// TIA Portal project "ConveyorSystem" (V16)

(* hardware
DEVICE "HMI_1"  KTP400 Comfort
   slot 0: "HMI_1"  KTP400 Comfort  6AV2 124-2DC01-0AX0  16.0.0.0
   slot 1: "HMI_RT_1"  KTP400 Comfort  6AV2 124-2DC01-0AX0  16.0.0.0
   slot 5: "HMI_1.IE_CP_1"  PROFINET Interface  16.0.0.0
      slot 1: "PROFINET Interface_1"  PROFINET Interface
         slot 1: "Port_1"  Port
   slot 7: "HMI_1.MPI/DP_CP_1"  MPI/DP Interface  16.0.0.0
DEVICE "S7-1200 station_1"  S7-1200 Station
   slot 0: "Rack_0"  S7-1200 Rack  Rack  V1.0
   slot 1: "PLC_1"  CPU 1217C DC/DC/DC  6ES7 217-1AG40-0XB0  V4.4
   slot 2: "DI 16x24VDC_1"  6ES7 221-1BH32-0XB0  V2.0
   slot 3: "DQ 16x24VDC_1"  SM 1222 DQ16 x 24VDC  6ES7 222-1BH32-0XB0  V2.0
*)

// ===== PLC "PLC_1"  CPU 1217C DC/DC/DC =====

VAR_GLOBAL   // PLC tag table "Default tag table"
   "System_Byte" AT %MB1 : Byte;
   "FirstScan" AT %M1.0 : Bool;
   "DiagStatusUpdate" AT %M1.1 : Bool;
   "AlwaysTRUE" AT %M1.2 : Bool;
   "AlwaysFALSE" AT %M1.3 : Bool;
   "Clock_Byte" AT %MB0 : Byte;
   "Clock_10Hz" AT %M0.0 : Bool;
   "Clock_5Hz" AT %M0.1 : Bool;
   "Clock_2.5Hz" AT %M0.2 : Bool;
   "Clock_2Hz" AT %M0.3 : Bool;
   "Clock_1.25Hz" AT %M0.4 : Bool;
   "Clock_1Hz" AT %M0.5 : Bool;
   "Clock_0.625Hz" AT %M0.6 : Bool;
   "Clock_0.5Hz" AT %M0.7 : Bool;
END_VAR

VAR_GLOBAL   // PLC tag table "Di"
   "Coveyor_Di" AT %I0.0 : "tyDi";
END_VAR

VAR_GLOBAL   // PLC tag table "Do"
   "ConveyorDo" AT %Q0.0 : "tyOutputs";
END_VAR

VAR_GLOBAL   // PLC tag table "SmemaIn"
   "SmemaIn-ReadyToSend" AT %I2.0 : Bool;
   "SmemaIn-ReadyToRecive" AT %Q2.0 : Bool;
END_VAR

VAR_GLOBAL   // PLC tag table "SmemaOut"
   "SmemaOut-ReadyToRecive" AT %I2.1 : Bool;
   "SmemaOut-ReadyToSend" AT %Q2.1 : Bool;
END_VAR

// folder: HmiExchange

TYPE "TyStopperHmiDataExchange"
   STRUCT
      FromPlcToHmi : Struct
         StopperUp : Bool;
         StopperDown : Bool;
         ProductPresent_BufferSpace : Bool;
         ProductPresent_Stopper : Bool;
      END_STRUCT;
      FromHmiToPlc : Struct
         DoStopperUp : Bool;
      END_STRUCT;
   END_STRUCT;
END_TYPE

TYPE "tyHmiMotorControl"
VERSION : 0.1
   STRUCT
      DataHmiToPlc : Struct
         doStartMotorForward : Bool;
      END_STRUCT;
      DataPlcToHmi : Struct
         MotorIsRuning : Bool;
      END_STRUCT;
   END_STRUCT;
END_TYPE

TYPE "TyModeControl"
VERSION : 0.1
   STRUCT
      StopPushButton : Bool;
      StartPusbutton : Bool;
      ManualMode : Bool;
      Reset : Bool;
   END_STRUCT;
END_TYPE

// folder: IO

TYPE "tyDi"
   STRUCT
      "IT-1-S1" : Bool;   // Input Trigger
      "B1-S1" : Bool;   // Buffer product detected
      "ST1-S1" : Bool;   // Stopper Up
      "ST1-S2" : Bool;   // Stopper Down
      "ST1-S3" : Bool;   // Stopper product detected
      "B2-S2" : Bool;   // Buffer product detected
      "ST2-S1" : Bool;   // Stopper Up
      "ST2-S2" : Bool;   // Stopper Down
      "ST2-S3" : Bool;   // Stopper product detected
      "IT2-S1" : Bool;   // Product Ready Acc
      "OT1-S1" : Bool;   // Output Trigger
      "M1-Runing" : Bool;   // Motor Forward Feedback
      MotorTemp_Ok : Bool;
      MotorProtection_Ok : Bool;
      "E-Stop_Ok" : Bool;
      AirSupply_Ok : Bool;
   END_STRUCT;
END_TYPE

TYPE "tyOutputs"
VERSION : 0.1
   STRUCT
      MotorForward : Bool;   // MotorForward
      "ST1-V1" : Bool;   // Stopper Valve
      "ST2-V1" : Bool;   // Stopper Valve
      ProductOnWorkPossition : Bool;
   END_STRUCT;
END_TYPE

// folder: (top level)

DATA_BLOCK "GVL"   // DB1
{ S7_Optimized_Access := 'TRUE' }
VERSION : 0.1
   VAR
      TestModeStruct : Struct
         TestMode : Bool;
      END_STRUCT;
      ScreenMode : Struct
         CurrentScreen : Int;
      END_STRUCT;
   END_VAR
   VAR RETAIN
      Parameters : Struct
         AccModeSellected : Bool;
         CurrentMode : Int;
      END_STRUCT;
   END_VAR
   VAR
      JobMailBox : Array[0..3] of Word;
      ScreenNumberHmiControl : Int;
      HmiCurrentScreenNumber : Array[0..4] of Word;
      CurrentScreen : Int;
   END_VAR
BEGIN
   JobMailBox[0] := 51;
   JobMailBox[2] := 0;
   JobMailBox[3] := 0;
END_DATA_BLOCK

// folder: DB

DATA_BLOCK "MainBlock_DB"   // DB2
{ S7_Optimized_Access := 'TRUE' }
VERSION : 0.1
// stored: InstanceOfName MainBlock
"MainBlock"
BEGIN
END_DATA_BLOCK

// folder: (top level)

ORGANIZATION_BLOCK "Main"   // OB1, LAD, ProgramCycle
TITLE = "Main Program Sweep (Cycle)"
{ S7_Optimized_Access := 'TRUE' }
VERSION : 0.1
   VAR_INPUT
      Initial_Call : Bool;   // Initial call of this OB
      Remanence : Bool;   // =True, if remanent data are available
   END_VAR
BEGIN

REGION Network 1
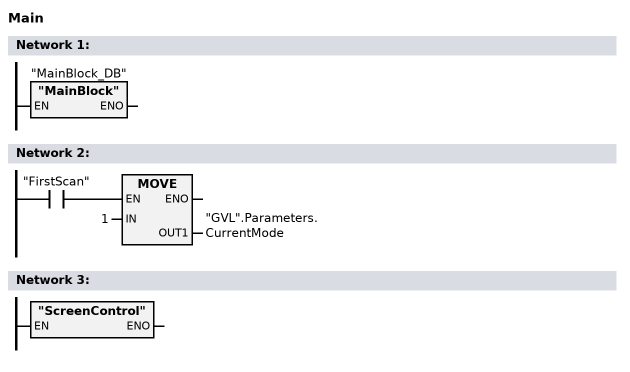
   RUNG wire#powerrail
      "MainBlock_DB"()
   END_RUNG
   // the same network as SCL:
   "MainBlock_DB"();   // "MainBlock"
END_REGION

REGION Network 2
   RUNG wire#powerrail
      Contact( "FirstScan" )
      Move(in := 1, out1 => "GVL".Parameters.CurrentMode)
   END_RUNG
   // the same network as SCL:
   IF "FirstScan" THEN "GVL".Parameters.CurrentMode := 1; END_IF;
END_REGION

REGION Network 3
   RUNG wire#powerrail
      "ScreenControl"()
   END_RUNG
   // the same network as SCL:
   "ScreenControl"();
END_REGION
END_ORGANIZATION_BLOCK

// folder: Devices

FUNCTION_BLOCK "Stopper"   // FB1, SCL
{ S7_Optimized_Access := 'TRUE' }
VERSION : 0.1
   VAR_INPUT
      TestMode : Bool;
      Di_Activate_StopperUp : Bool;
      Di_StopperSensorUp : Bool;
      Di_StopperSensorDown : Bool;
      Di_StopperSensorProductDetected : Bool;
      Di_BufferrSensorProductDetected : Bool;
      ManualMode : Bool;
   END_VAR
   VAR_OUTPUT
      Do_Fault : Bool;
      Do_OutputSolenoidValve_Up : Bool;
      Do_StopperIsUp : Bool;
      Do_StopperIsDown : Bool;
      Do_ProductDetectedStopper : Bool;
      Do_ProductDetectedBuffer : Bool;
   END_VAR
   VAR
      HmiStopperExchange : "TyStopperHmiDataExchange";
      StopperUpFault : TON_TIME;
      StopperDownFault : TON_TIME;
   END_VAR
BEGIN
   //=============================================================================
   // Dmitri Raihtsaum - Copyright 2024
   // Created By: Dmitri Raihtsaum
   //-----------------------------------------------------------------------------
   // Tested with:   6ES7 217-1AG40-0XB0
   // Engineering:   TIA Portal V16
   // Functionality:  Stopper Controll fucntion block
   // Date: 13.10.2024
   // Rev 0.1
   //=============================================================================

   //Manual Auto Control Switch
   IF #ManualMode THEN
       IF #HmiStopperExchange.FromHmiToPlc.DoStopperUp THEN
           #Do_OutputSolenoidValve_Up := TRUE;
       ELSE
           #Do_OutputSolenoidValve_Up := FALSE;
       END_IF;
   ELSE
       IF #Di_Activate_StopperUp THEN
           #Do_OutputSolenoidValve_Up := TRUE;
       ELSE
           #Do_OutputSolenoidValve_Up := FALSE;
       END_IF;
   END_IF;

   //Fault Control
   IF #TestMode THEN
       #StopperUpFault(IN := FALSE,
                       PT := t#0ms);
       #StopperDownFault(IN := FALSE,
                         PT := t#0ms);
   ELSE
       #StopperUpFault(IN := #Di_Activate_StopperUp AND NOT #Do_StopperIsUp,
                       PT := t#2s);
       #StopperDownFault(IN := NOT #Di_Activate_StopperUp AND NOT #Do_StopperIsDown,
                         PT := t#2s);
   END_IF;

   //Fault Control
   IF #StopperDownFault.Q OR #StopperUpFault.Q THEN
       #Do_Fault := TRUE;
   ELSE
       #Do_Fault := FALSE;
   END_IF;

   //Do
   IF #TestMode THEN
       #Do_StopperIsUp := #Do_OutputSolenoidValve_Up;
       #Do_StopperIsDown := NOT  #Do_OutputSolenoidValve_Up;
   ELSE
       #Do_StopperIsUp := #Di_StopperSensorUp;
       #Do_StopperIsDown := #Di_StopperSensorDown;
   END_IF;
   #Do_ProductDetectedStopper := #Di_StopperSensorProductDetected;
   #Do_ProductDetectedBuffer := #Di_BufferrSensorProductDetected;

   //Hmi
   #HmiStopperExchange.FromPlcToHmi.StopperUp := #Do_StopperIsUp;
   #HmiStopperExchange.FromPlcToHmi.StopperDown := #Do_StopperIsDown;
   #HmiStopperExchange.FromPlcToHmi.ProductPresent_BufferSpace := #Di_StopperSensorProductDetected;
   #HmiStopperExchange.FromPlcToHmi.ProductPresent_Stopper := #Di_BufferrSensorProductDetected;

   //=============================================================================
   //END
   //=============================================================================
END_FUNCTION_BLOCK

FUNCTION_BLOCK "MotorControl"   // FB2, SCL
{ S7_Optimized_Access := 'TRUE' }
VERSION : 0.1
   VAR_INPUT
      TestMode : Bool;
      ManualMode : Bool;
      Di_doStartMotorForward : Bool;
      Di_MotorForwardFeedback : Bool;
      Di_MotorTemp_Ok : Bool;
      Di_MotorProtection_Ok : Bool;
   END_VAR
   VAR_OUTPUT
      Do_Fault : Bool;
      Do_StartMotorForward : Bool;
      Do_MotorIsRuning : Bool;
   END_VAR
   VAR
      Hmi_MotorDataExchange : "tyHmiMotorControl";
      MotorRunFault : TON_TIME;
      MotorStopFault : TON_TIME;
   END_VAR
BEGIN
   //=============================================================================
   // Dmitri Raihtsaum - Copyright 2024
   // Created By: Dmitri Raihtsaum
   //-----------------------------------------------------------------------------
   // Tested with:   6ES7 217-1AG40-0XB0 
   // Engineering:   TIA Portal V16
   // Functionality:  Motor Controll fucntion block
   // Date: 13.10.2024
   // Rev 0.1
   //=============================================================================

   //Manual Auto Control Switch
   IF #ManualMode THEN
       IF #Hmi_MotorDataExchange.DataHmiToPlc.doStartMotorForward THEN
           #Do_StartMotorForward := TRUE;
       ELSE
           #Do_StartMotorForward := FALSE;
       END_IF;
   ELSE
       IF #Di_doStartMotorForward THEN
           #Do_StartMotorForward := TRUE;
       ELSE
           #Do_StartMotorForward := FALSE;
       END_IF;
   END_IF;
   //Fault Control
   IF #TestMode THEN
       #MotorRunFault(IN := FALSE,
                      PT := T#2s);
       #MotorStopFault(IN := FALSE,
                       PT := T#2s);
   ELSE
       #MotorRunFault(IN := #Di_doStartMotorForward AND NOT #Di_MotorForwardFeedback,
                      PT := T#2s);
       #MotorStopFault(IN := NOT #Di_doStartMotorForward AND #Di_MotorForwardFeedback,
                       PT := T#2s);
   END_IF;
   //Fault Control
   IF NOT #TestMode THEN
       #Do_Fault := NOT #Di_MotorTemp_Ok OR NOT #Di_MotorProtection_Ok OR #MotorRunFault.Q OR #MotorStopFault.Q;
   ELSE
       #Do_Fault := FALSE;
   END_IF;
   //Motor Feedback 
   IF NOT #TestMode THEN
       #Do_MotorIsRuning := #Di_MotorForwardFeedback;
   ELSE
       #Do_MotorIsRuning := #Do_StartMotorForward;
   END_IF;

   #Hmi_MotorDataExchange.DataPlcToHmi.MotorIsRuning := #Do_MotorIsRuning;

   //=============================================================================
   //END
   //=============================================================================
END_FUNCTION_BLOCK

// folder: Logic

FUNCTION_BLOCK "SystemControl"   // FB3, SCL
{ S7_Optimized_Access := 'TRUE' }
VERSION : 0.1
   VAR_INPUT
      Di_ReadyToStop : Bool;
      Di_ExternalFault : Bool;
   END_VAR
   VAR_OUTPUT
      SystemStateOutput : Int;
      Do_ManualMode : Bool;
      Do_Reset : Bool;
   END_VAR
   VAR
      CurrentState : Int;
      HmiSystemControl : "TyModeControl";
      StopTimer : TON_TIME;
   END_VAR
BEGIN
   //=============================================================================
   // Dmitri Raihtsaum - Copyright 2024
   // Created By: Dmitri Raihtsaum
   //-----------------------------------------------------------------------------
   // Tested with:   6ES7 215-1AG40-0XB0
   // Engineering:   TIA Portal V16
   // Functionality:  Mode Control 
   // Date: 13.10.2024
   // Rev 0.1
   //=============================================================================

   CASE #CurrentState OF
       0:  // Var Init
           IF "FirstScan" OR #HmiSystemControl.Reset THEN
               #CurrentState := 1;
           END_IF;

       1:  // Stop
           IF #HmiSystemControl.StartPusbutton THEN
               #CurrentState := 2;
           END_IF;

       2: //AutoRun
           IF (#HmiSystemControl.StopPushButton AND NOT #Di_ReadyToStop) THEN
               #CurrentState := 3;
           ELSIF (#HmiSystemControl.StopPushButton AND #Di_ReadyToStop) THEN
               #CurrentState := 1;
           END_IF;

       3: //AutoStop
           IF #Di_ReadyToStop OR #StopTimer.Q THEN
               #CurrentState := 1;
           END_IF;
   END_CASE;

   #StopTimer(IN := #HmiSystemControl.StopPushButton,
              PT := T#2s);

   IF #Di_ExternalFault THEN
       #CurrentState := 0;
   END_IF;
   #Do_ManualMode := #HmiSystemControl.ManualMode;

   #SystemStateOutput := #CurrentState;

   //=============================================================================
   //END
   //=============================================================================
END_FUNCTION_BLOCK

FUNCTION_BLOCK "MainBlock"   // FB4, SCL
{ S7_Optimized_Access := 'TRUE' }
VERSION : 0.1
   VAR
      MainLogic_Instance : "MainLogic";
   END_VAR
BEGIN
   //=============================================================================
   // Dmitri Raihtsaum - Copyright 2024
   // Created By: Dmitri Raihtsaum
   //-----------------------------------------------------------------------------
   // Tested with:   6ES7 217-1AG40-0XB0 
   // Engineering:   TIA Portal V16
   // Functionality:  Main Block Logic
   // Date: 13.10.2024
   // Rev 0.1
   //=============================================================================
   //
   CASE "GVL".Parameters.CurrentMode OF
       1:  // Mode 1
           #MainLogic_Instance(Di_Input:="Coveyor_Di",
                               "SmemaIn-ReadyToSend":="SmemaIn-ReadyToSend",
                               "SmemaOut-ReadyToRecive":="SmemaOut-ReadyToRecive",
                               TestMode:="GVL".TestModeStruct.TestMode,
                               Do_Output=>"ConveyorDo",
                               "SmemaIn-ReadyToRecive"=>"SmemaIn-ReadyToRecive",
                               "SmemaOut-ReadyToSend"=>"SmemaOut-ReadyToSend");

       2:  // Mode 2
           ;

   END_CASE;

   //=============================================================================
   //END
   //=============================================================================
END_FUNCTION_BLOCK

FUNCTION_BLOCK "MainLogic"   // FB5, SCL
{ S7_Optimized_Access := 'TRUE' }
VERSION : 0.1
   VAR_INPUT
      Di_Input : "tyDi";
      "SmemaIn-ReadyToSend" : Bool;
      "SmemaOut-ReadyToRecive" : Bool;
      TestMode : Bool;
      OperatorOrRobotAcknowledge_Setting : Bool;
   END_VAR
   VAR_OUTPUT
      Do_Output : "tyOutputs";
      "SmemaIn-ReadyToRecive" : Bool := false;
      "SmemaOut-ReadyToSend" : Bool := false;
      GlobalReset : Bool := false;
      Alarms0 : Word := 16#0;
   END_VAR
   VAR
      CurrentState : Int;
      Stopper_1 : "Stopper";
      Stopper_2 : "Stopper";
      MotorControl_1 : "MotorControl";
      SystemControl_Instance : "SystemControl";
      StepTimer1 : TON_TIME;
      StepTimer2 : TON_TIME;
      OutputTriggerDelay : TOF_TIME;
   END_VAR
BEGIN
   //=============================================================================
   // Dmitri Raihtsaum - Copyright 2024
   // Created By: Dmitri Raihtsaum
   //-----------------------------------------------------------------------------
   // Tested with:   6ES7 217-1AG40-0XB0 
   // Engineering:   TIA Portal V16
   // Functionality:  Main Logic
   // Date: 13.10.2024
   // Rev 0.1
   //=============================================================================

   CASE #CurrentState OF
       0:  // Var Init
           #StepTimer1(IN:=FALSE,
                       PT:=T#0ms);
           #StepTimer2(IN:=FALSE,
                       PT:=T#0ms);
           #"SmemaIn-ReadyToRecive" := FALSE;
           #"SmemaOut-ReadyToSend" := FALSE;
           #Do_Output.ProductOnWorkPossition := FALSE;
           #Stopper_1.Di_Activate_StopperUp := TRUE;
           #Stopper_2.Di_Activate_StopperUp := TRUE;
           #MotorControl_1.Di_doStartMotorForward := FALSE;
           #SystemControl_Instance.Di_ReadyToStop := TRUE;
           IF #SystemControl_Instance.SystemStateOutput = 2 THEN
               #CurrentState := 1;
           END_IF;

       1:  // Stopper Test 
           #Stopper_1.Di_Activate_StopperUp := FALSE;
           #Stopper_2.Di_Activate_StopperUp := FALSE;
           #StepTimer1(IN := TRUE,
                       PT := T#700ms);
           #StepTimer2(IN := FALSE,
                       PT := T#0ms);
           IF #StepTimer1.Q THEN
               #CurrentState := 2;
           END_IF;
       2: // Stopper Test 
           #StepTimer1(IN := FALSE,
                       PT := T#0ms);
           #StepTimer2(IN := TRUE,
                       PT := T#500ms);
           #Stopper_1.Di_Activate_StopperUp := TRUE;
           #Stopper_2.Di_Activate_StopperUp := TRUE;
           IF #StepTimer2.Q THEN
               #CurrentState := 3;
           END_IF;

       3:// Stopper Test 
           #StepTimer1(IN := TRUE,
                       PT := T#1s);
           #StepTimer2(IN := FALSE,
                       PT := T#0ms);
           #MotorControl_1.Di_doStartMotorForward := TRUE;
           IF #StepTimer1.Q THEN
               #CurrentState := 10;
           END_IF;

       6: //Idle 
           #StepTimer1(IN := FALSE,
                       PT := T#0ms);
           #StepTimer2(IN := FALSE,
                       PT := T#0ms);
           #"SmemaIn-ReadyToRecive" := FALSE;
           #"SmemaOut-ReadyToSend" := FALSE;
           #Do_Output.ProductOnWorkPossition := FALSE;
           #Stopper_1.Di_Activate_StopperUp := TRUE;
           #Stopper_2.Di_Activate_StopperUp := TRUE;
           #MotorControl_1.Di_doStartMotorForward := FALSE;
           #SystemControl_Instance.Di_ReadyToStop := TRUE;
           // Product move sellection 
           IF #SystemControl_Instance.SystemStateOutput = 2 THEN
               IF (#"SmemaIn-ReadyToSend" OR #Di_Input."IT-1-S1") AND NOT #Stopper_1.Do_ProductDetectedStopper THEN
                   #CurrentState := 10;
               ELSIF NOT #Stopper_2.Do_ProductDetectedStopper AND #Stopper_1.Do_ProductDetectedStopper THEN
                   #CurrentState := 30;
               ELSIF #OperatorOrRobotAcknowledge_Setting AND #Stopper_2.Do_ProductDetectedStopper AND #"SmemaOut-ReadyToRecive" AND #Di_Input."IT2-S1"
               THEN
                   #CurrentState := 40;
               ELSIF NOT #OperatorOrRobotAcknowledge_Setting AND #Stopper_2.Do_ProductDetectedStopper AND #"SmemaOut-ReadyToRecive" THEN
                   #CurrentState := 40;
               END_IF;
           END_IF;


       10: // Pass sellection - Go to buffer 1 - or move to buffer 2 
           #SystemControl_Instance.Di_ReadyToStop := FALSE;
           IF NOT #Stopper_2.Do_ProductDetectedStopper AND NOT #"SmemaOut-ReadyToRecive" AND NOT #OperatorOrRobotAcknowledge_Setting THEN
               #CurrentState := 20;
           ELSIF NOT #Stopper_2.Do_ProductDetectedStopper AND #"SmemaOut-ReadyToRecive" AND NOT #OperatorOrRobotAcknowledge_Setting THEN
               #CurrentState := 50;
           ELSE
               #CurrentState := 11;
           END_IF;

       11: // Move to stopper 1
           #SystemControl_Instance.Di_ReadyToStop := FALSE;
           #StepTimer1(IN := FALSE,
                       PT := T#0ms);
           #StepTimer2(IN := FALSE,
                       PT := T#0ms);
           #"SmemaIn-ReadyToRecive" := TRUE;
           #Stopper_1.Di_Activate_StopperUp := TRUE;
           #MotorControl_1.Di_doStartMotorForward := TRUE;
           IF #Stopper_1.Do_ProductDetectedStopper THEN
               #CurrentState := 12;
           END_IF;

       12: // Stop product to stopper 1
           #StepTimer1(IN := TRUE,
                       PT := T#1s);
           #StepTimer2(IN := FALSE,
                       PT := T#0ms);
           #"SmemaIn-ReadyToRecive" := FALSE;
           #Stopper_1.Di_Activate_StopperUp := TRUE;
           #MotorControl_1.Di_doStartMotorForward := FALSE;
           IF #StepTimer1.Q THEN
               #CurrentState := 6;
           END_IF;

       20: // Move to stopper 2
           #SystemControl_Instance.Di_ReadyToStop := FALSE;
           #StepTimer1(IN := FALSE,
                       PT := T#0ms);
           #StepTimer2(IN := FALSE,
                       PT := T#0ms);
           #"SmemaIn-ReadyToRecive" := TRUE;
           #Stopper_1.Di_Activate_StopperUp := FALSE;
           #Stopper_2.Di_Activate_StopperUp := TRUE;
           #MotorControl_1.Di_doStartMotorForward := TRUE;
           IF #Stopper_2.Do_ProductDetectedStopper THEN
               #CurrentState := 21;
           END_IF;

       21: // Stop product to stopper 2
           #StepTimer1(IN := TRUE,
                       PT := T#1s);
           #StepTimer2(IN := FALSE,
                       PT := T#0ms);
           #"SmemaIn-ReadyToRecive" := FALSE;
           #Stopper_1.Di_Activate_StopperUp := TRUE;
           #Stopper_2.Di_Activate_StopperUp := TRUE;
           #MotorControl_1.Di_doStartMotorForward := FALSE;
           IF #StepTimer1.Q THEN
               #CurrentState := 6;
           END_IF;

       30 : //  Buffer 1 to buffer 2 transit 
           #SystemControl_Instance.Di_ReadyToStop := FALSE;
           #StepTimer1(IN := FALSE,
                       PT := T#0ms);
           #StepTimer2(IN := FALSE,
                       PT := T#0ms);
           #Stopper_1.Di_Activate_StopperUp := FALSE;
           #Stopper_2.Di_Activate_StopperUp := TRUE;
           #MotorControl_1.Di_doStartMotorForward := TRUE;
           IF #Stopper_2.Do_ProductDetectedStopper THEN
               #CurrentState := 31;
           END_IF;

       31: // Buffer 1 to buffer 2 transit 
           #StepTimer1(IN := TRUE,
                       PT := T#1s);
           #StepTimer2(IN := FALSE,
                       PT := T#0ms);
           #Stopper_1.Di_Activate_StopperUp := TRUE;
           #Stopper_2.Di_Activate_StopperUp := TRUE;
           #MotorControl_1.Di_doStartMotorForward := FALSE;
           IF #StepTimer1.Q THEN
               #CurrentState := 6;
           END_IF;

       40 : // Out Transit 
           #SystemControl_Instance.Di_ReadyToStop := FALSE;
           #OutputTriggerDelay(IN:=FALSE,
                               PT:=T#0ms);
           #Stopper_2.Di_Activate_StopperUp := FALSE;
           #MotorControl_1.Di_doStartMotorForward := TRUE;
           IF #Di_Input."OT1-S1" THEN
               #CurrentState := 41;
           END_IF;

       41: //  Out Transit 
           #OutputTriggerDelay(IN := #Di_Input."OT1-S1",
                               PT := T#15s);
           IF #OutputTriggerDelay.ET > T#6s THEN
               #CurrentState := 6;
           END_IF;


       50: // Transit withour stopper 
           #SystemControl_Instance.Di_ReadyToStop := FALSE;
           #StepTimer1(IN := FALSE,
                       PT := T#0ms);
           #StepTimer2(IN := FALSE,
                       PT := T#0ms);
           #OutputTriggerDelay(IN := FALSE,
                               PT := T#0ms);
           #Stopper_1.Di_Activate_StopperUp := FALSE;
           #Stopper_2.Di_Activate_StopperUp := FALSE;
           #MotorControl_1.Di_doStartMotorForward := TRUE;
           IF #Di_Input."OT1-S1" THEN
               #CurrentState := 51;
           END_IF;

       51: // Transit withour stopper 
           #OutputTriggerDelay(IN := #Di_Input."OT1-S1",
                               PT := T#15s);
           IF #OutputTriggerDelay.ET > T#6s THEN
               #CurrentState := 6;
           END_IF;


   END_CASE;

   IF #SystemControl_Instance.CurrentState < 2 THEN
       #CurrentState := 6;
   END_IF;

   #Stopper_1(TestMode:=#TestMode,
              Di_StopperSensorUp:=#Di_Input."ST1-S1",
              Di_StopperSensorDown:=#Di_Input."ST1-S2",
              Di_StopperSensorProductDetected:=#Di_Input."ST1-S3",
              Di_BufferrSensorProductDetected:=#Di_Input."B1-S1",
              ManualMode:=#SystemControl_Instance.Do_ManualMode,
              Do_OutputSolenoidValve_Up=>#Do_Output."ST1-V1");
   #Stopper_2(TestMode:=#TestMode,
              Di_StopperSensorUp:=#Di_Input."ST2-S1",
              Di_StopperSensorDown:=#Di_Input."ST2-S2",
              Di_StopperSensorProductDetected:=#Di_Input."ST2-S3",
              Di_BufferrSensorProductDetected:=#Di_Input."B2-S2",
              ManualMode:=#SystemControl_Instance.Do_ManualMode,
              Do_OutputSolenoidValve_Up=>#Do_Output."ST2-V1");
   #MotorControl_1(TestMode:=#TestMode,
                   ManualMode:=#SystemControl_Instance.Do_ManualMode,
                   Di_MotorForwardFeedback:=#Di_Input."M1-Runing",
                   Di_MotorTemp_Ok:=#Di_Input.MotorTemp_Ok,
                   Di_MotorProtection_Ok:=#Di_Input.MotorProtection_Ok,
                   Do_StartMotorForward=>#Do_Output.MotorForward);
   #SystemControl_Instance();

   REGION Alarms
       IF #TestMode THEN
           #Alarms0.%X0 := FALSE;
           #Alarms0.%X1 := FALSE;
           #Alarms0.%X2 := FALSE;
           #Alarms0.%X3 := FALSE;
           #Alarms0.%X4 := FALSE;
           #Alarms0.%X5 := FALSE;
           #Alarms0.%X6 := FALSE;
           //  #Alarms0.%X7 :=
       ELSE

           #Alarms0.%X0 := NOT #Di_Input.MotorTemp_Ok;
           #Alarms0.%X1 := NOT #Di_Input.MotorProtection_Ok;
           #Alarms0.%X2 := NOT #Di_Input."E-Stop_Ok";
           #Alarms0.%X3 := NOT #Di_Input.AirSupply_Ok;
           #Alarms0.%X4 := #Stopper_1.Do_Fault;
           #Alarms0.%X5 := #Stopper_1.Do_Fault;
           #Alarms0.%X6 := #MotorControl_1.Do_Fault;
           //  #Alarms0.%X7 :=
       END_IF;

   END_REGION
   //=============================================================================
   //END
   //=============================================================================
END_FUNCTION_BLOCK

FUNCTION "ScreenControl" : Void   // FC1, SCL
{ S7_Optimized_Access := 'TRUE' }
VERSION : 0.1
BEGIN
   //=============================================================================
   // Dmitri Raihtsaum - Copyright 2024
   // Created By: Dmitri Raihtsaum
   //-----------------------------------------------------------------------------
   // Tested with:   6ES7 217-1AG40-0XB0 
   // Engineering:   TIA Portal V16
   // Functionality:  Screen Control
   // Date: 13.10.2024
   // Rev 0.1
   //=============================================================================

   "GVL".CurrentScreen := WORD_TO_INT("GVL".HmiCurrentScreenNumber[1]); // Recive information from current screen 
   "GVL".ScreenNumberHmiControl := "GVL".Parameters.CurrentMode * 10; // Prepare variable to activate screen

   IF "GVL".CurrentScreen / 10 <> "GVL".Parameters.CurrentMode THEN // Compare current screen and current mode
       "GVL".JobMailBox[1] := INT_TO_WORD("GVL".ScreenNumberHmiControl); // Send screen number to hmi to change screen 
       "GVL".JobMailBox[0] := 16#33; // Jobmailbox adress
       "GVL".JobMailBox[2] := 16#00; // Not used 
       "GVL".JobMailBox[3] := 16#00; // Not used 
   END_IF;

   //=============================================================================
   //END
   //=============================================================================
END_FUNCTION

(* ===== HMI "HMI_RT_1" =====
system functions are stored by id; their names below are inferred from use
connection "HMI_Connection_1": ETHERNET, S7_1200_OMS

HMI tags "Di"
   "Di" : tyDi = PLC Coveyor_Di AT %I0.0, 1 s

HMI tags "Do"
   "Do" : tyOutputs = PLC ConveyorDo AT %Q0.0, 1 s

HMI tags "SmemaIn"
   "SmemaIn-ReadyToRecive" : Bool = PLC "SmemaIn-ReadyToRecive" AT %Q2.0, 1 s
   "SmemaIn-ReadyToSend" : Bool = PLC "SmemaIn-ReadyToSend" AT %I2.0, 1 s

HMI tags "SmemaOut"
   "SmemaOut-ReadyToRecive" : Bool = PLC "SmemaOut-ReadyToRecive" AT %I2.1, 1 s
   "SmemaOut-ReadyToSend" : Bool = PLC "SmemaOut-ReadyToSend" AT %Q2.1, 1 s

HMI tags "SystemControl"
   "HmiSystemControl" : TyModeControl = PLC MainBlock_DB.MainLogic_Instance.SystemControl_Instance.HmiSystemControl, 1 s

HMI tags "Stoppers"
   "HmiStopperExchange1" : TyStopperHmiDataExchange = PLC MainBlock_DB.MainLogic_Instance.Stopper_1.HmiStopperExchange, 1 s
   "HmiStopperExchange2" : TyStopperHmiDataExchange = PLC MainBlock_DB.MainLogic_Instance.Stopper_2.HmiStopperExchange, 1 s

HMI tags "Motors"
   "Hmi_MotorDataExchange" : tyHmiMotorControl = PLC MainBlock_DB.MainLogic_Instance.MotorControl_1.Hmi_MotorDataExchange, 1 s

HMI tags "Parameters"
   "CurrentModeSellection" : Int = PLC GVL.Parameters.CurrentMode, 1 s
   "AccModeActivated" : Bool = PLC GVL.Parameters.AccModeSellected AT %DB1.DBW0, 1 s

HMI tags "SystemData"
   "SystemMode" : Int = PLC MainBlock_DB.MainLogic_Instance.SystemControl_Instance.SystemStateOutput, 1 s

HMI tags "Alarm0"
   "Alarm0" : Word = PLC MainBlock_DB.MainLogic_Instance.Alarms0 AT %DB1.DBW0, 1 s

discrete alarms
   1: 'Motor Temperature fault', class Errors, trigger "Alarm0" bit 0
   2: 'Motor Protection Triggered', class Errors, trigger "Alarm0" bit 1
   3: 'E-Stop Triggred', class Errors, trigger "Alarm0" bit 2
   4: 'Air Sypply Fault', class Errors, trigger "Alarm0" bit 3
   5: 'Stopper 1 Fault', class Errors, trigger "Alarm0" bit 4
   6: 'Stopper 2 Fault', class Errors, trigger "Alarm0" bit 5
   7: 'Motor Fault', class Errors, trigger "Alarm0" bit 6

Template "Template_1" 480x272
   Button "Template_Button_1" at 12,7 size 96x32; TextOff 'Start'
      ObjectEnable <- "ManualMode"
      on Press: function_b14e0dd5("StartPusbutton", 0); ResetBit("doStartMotorForward"); ResetBit("DoStopperUp"); ResetBit("DoStopperUp")
      Appearance <- "SystemMode"
   Button "Template_Button_2" at 124,7 size 96x32; TextOff 'Stop'
      on Press: function_b14e0dd5("StopPushButton", 0)
      Appearance <- "SystemMode"
   Button "Template_Button_3" at 237,7 size 96x32; TextOff 'Reset'
      on Press: function_b14e0dd5("Reset", 0)
      Appearance <- "Reset"
   Button "Template_Button_4" at 376,7 size 96x32; TextOff 'Menu'
      on Click: ActivateScreen("Menu", 0)

screen "RootMode1" 480x272, template "Template_1"
   Circle "Circle_1" at 421,84 size 34x34
      Appearance <- "MotorIsRuning"
   Rectangle "Rectangle_2" at 129,133 size 15x43
      Visibility <- "StopperUp"
   Rectangle "Rectangle_3" at 129,180 size 15x43
      Visibility <- "StopperDown"
   Rectangle "Rectangle_4" at 294,133 size 15x43
      Visibility <- "StopperUp"
   Rectangle "Rectangle_5" at 294,180 size 15x43
      Visibility <- "StopperDown"
   TextField "Text field_1" at 73,96 size 65x20; Text 'Buffer 1'
   TextField "Text field_2" at 229,98 size 65x20; Text 'Buffer 2'
   Circle "Circle_2" at 272,141 size 20x20
      Appearance <- "ST2-S3"
   Circle "Circle_3" at 231,141 size 20x20
      Appearance <- "B2-S2"
   Circle "Circle_4" at 106,141 size 20x20
      Appearance <- "ST1-S3"
   Circle "Circle_5" at 67,141 size 20x20
      Appearance <- "B1-S1"
   Circle "Circle_6" at 11,170 size 20x20
      Appearance <- "SmemaIn-ReadyToSend"
   Circle "Circle_7" at 11,197 size 20x20
      Appearance <- "IT-1-S1"
   TextField "Text field_3" at 28,170 size 113x20; Text 'Ready to Send'
   TextField "Text field_4" at 29,197 size 103x20; Text 'Input Trigger'
   TextField "Text field_5" at 430,91 size 17x20; Text 'M'
   Circle "Circle_8" at 446,170 size 20x20
      Appearance <- "SmemaOut-ReadyToRecive"
   Circle "Circle_9" at 446,197 size 20x20
      Appearance <- "OT1-S1"
   TextField "Text field_6" at 328,170 size 126x20; Text 'Ready to Recive'
   TextField "Text field_7" at 328,197 size 114x20; Text 'Output Trigger'
   Circle "Circle_10" at 274,234 size 20x20
      Appearance <- "IT2-S1"
   TextField "Text field_8" at 168,234 size 104x20; Text 'Operator Acc'

screen "RootMode2" 480x272
   TextField "Text field_1" at 146,122 size 58x20; Text 'Mode 2'

screen "Parameters" 480x272
   Button "Button_1" at 2,236 size 96x32; TextOff 'Back'
      on Click: function_efd93a16()
   IOField "I/O field_1" at 239,95 size 96x32; FormatPattern 99
      ProcessValue <- "CurrentModeSellection"
   TextField "Text field_1" at 179,101 size 44x20; Text 'Mode'
   Button "Button_2" at 179,153 size 190x32; TextOff 'Opeator ACC Option'
      on Click: InvertBit("AccModeActivated")
      Appearance <- "AccModeActivated"

screen "Menu" 480x272, template "Template_1"
   Button "Button_1" at 136,87 size 192x32; TextOff 'Parameters'
      on Click: ActivateScreen("Parameters", 0)
   Button "Button_2" at 136,135 size 192x32; TextOff 'ManualMode'
      on Click: ActivateScreen("ManualMode", 0)
   Button "Button_3" at 2,236 size 96x32; TextOff 'Back'
      on Click: function_efd93a16()

screen "ManualMode" 480x272, template "Template_1"
   Button "Button_1" at 2,236 size 96x32; TextOff 'Back'
      on Click: function_efd93a16()
   Button "Button_2" at 11,68 size 96x32; TextOff 'Manual Mode'
      on Click: InvertBit("ManualMode")
      Appearance <- "ManualMode"
      on Press: ResetBit("doStartMotorForward"); ResetBit("DoStopperUp"); ResetBit("DoStopperUp")
      ObjectEnable <- "SystemMode"
   Button "Button_3" at 11,116 size 96x32; TextOff 'Motor'
      Appearance <- "doStartMotorForward"
      on Click: InvertBit("doStartMotorForward")
   Button "Button_4" at 158,116 size 96x32; TextOff 'Stopper 1'
      on Click: InvertBit("DoStopperUp")
      Appearance <- "DoStopperUp"
   Button "Button_5" at 158,161 size 96x32; TextOff 'Stopper 2'
      on Click: InvertBit("DoStopperUp")
      Appearance <- "DoStopperUp"
*)